FUNCTION_BLOCK Model (* Composite Function Block Type *)
  (* Standard: 61499-2 *)
  (* Version 0.0, 6/17/2016, Andrei, nxtControl GmbH, template *)
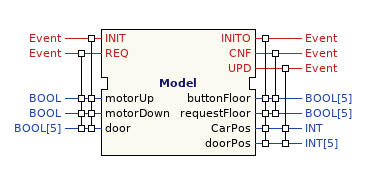
  EVENT_INPUT
    INIT WITH motorUp, motorDown, door; (* Initialization Request *)
    REQ WITH motorUp, motorDown, door; (* Normal Execution Request *)
  END_EVENT
  EVENT_OUTPUT
    INITO WITH buttonFloor, requestFloor, CarPos, doorPos; (* Initialization Confirm *)
    CNF WITH buttonFloor, requestFloor; (* Execution Confirmation *)
    UPD WITH CarPos, doorPos;
  END_EVENT
  VAR_INPUT
    motorUp : BOOL; (* Input event qualifier *)
    motorDown : BOOL;
    door : ARRAY [0..4] OF BOOL;
  END_VAR
  VAR_OUTPUT
    buttonFloor : ARRAY [0..4] OF BOOL; (* Output event qualifier *)
    requestFloor : ARRAY [0..4] OF BOOL;
    CarPos : INT;
    doorPos : ARRAY [0..4] OF INT;
  END_VAR
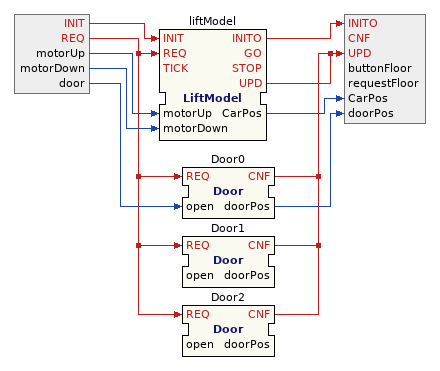
  FBS
    liftModel : LiftModel;
    Door0 : Door;
    Door1 : Door;
    Door2 : Door;
  END_FBS
  EVENT_CONNECTIONS
    INIT TO liftModel.INIT;
    REQ TO liftModel.REQ;
    liftModel.UPD TO UPD;
    liftModel.INITO TO INITO;
    Door0.CNF TO UPD;
    REQ TO Door0.REQ;
    Door1.CNF TO UPD;
    Door2.CNF TO UPD;
    REQ TO Door1.REQ;
    REQ TO Door2.REQ;
  END_CONNECTIONS
  DATA_CONNECTIONS
    motorUp TO liftModel.motorUp;
    motorDown TO liftModel.motorDown;
    liftModel.CarPos TO CarPos;
    Door0.doorPos TO doorPos;
    door TO Door0.open;
  END_CONNECTIONS
END_FUNCTION_BLOCK
